// TIA Portal V17 export
// export: Created 2023-12-22T15:05:34.1188852Z, ExportSetting WithDefaults, DisplayName Totally Integrated Automation Portal, DisplayVersion V17, DisplayName TIA Portal Openness, DisplayVersion V17, DisplayName TIA Portal Version Control Interface, DisplayVersion V17, DisplayName STEP 7 Professional, DisplayVersion V17, DisplayName STEP 7 Safety, DisplayVersion V17, DisplayName WinCC Advanced, DisplayVersion V17
DATA_BLOCK "DB_OUT"   // DB102
{ S7_Optimized_Access := 'FALSE' }
VERSION : 0.1
// stored: AutoNumber false, DBAccessibleFromOPCUA true, IsOnlyStoredInLoadMemory false, IsWriteProtectedInAS false
   VAR
      AI_FT_007 { S7_SetPoint := 'True'} : "Out_AI";
      AI_FT_008 { S7_SetPoint := 'True'} : "Out_AI";
      AI_FT_009 { S7_SetPoint := 'True'} : "Out_AI";
      AI_FT_010 { S7_SetPoint := 'True'} : "Out_AI";
      AI_LT_014 { S7_SetPoint := 'True'} : "Out_AI";
      AI_LT_015 { S7_SetPoint := 'True'} : "Out_AI";
      AI_LT_016 { S7_SetPoint := 'True'} : "Out_AI";
      AI_LT_019 { S7_SetPoint := 'True'} : "Out_AI";
      AI_PT_001 { S7_SetPoint := 'True'} : "Out_AI";
      AI_PT_002 { S7_SetPoint := 'True'} : "Out_AI";
      AI_PT_003 { S7_SetPoint := 'True'} : "Out_AI";
      AI_PT_004 { S7_SetPoint := 'True'} : "Out_AI";
      AI_PT_005 { S7_SetPoint := 'True'} : "Out_AI";
      AI_PT_006 { S7_SetPoint := 'True'} : "Out_AI";
      Z_GVM_020 { S7_SetPoint := 'True'} : "Out_Z";
      Z_GVM_021 { S7_SetPoint := 'True'} : "Out_Z";
      Z_GVM_022 { S7_SetPoint := 'True'} : "Out_Z";
      Z_GCM_023 { S7_SetPoint := 'True'} : "Out_Z";
      Z_GCM_024 { S7_SetPoint := 'True'} : "Out_Z";
      Z_GCM_025 { S7_SetPoint := 'True'} : "Out_Z";
      XVS_026 { S7_SetPoint := 'True'} : "InOut_DO";
      XVS_027 { S7_SetPoint := 'True'} : "InOut_DO";
      XVS_028 { S7_SetPoint := 'True'} : "InOut_DO";
      XVS_029 { S7_SetPoint := 'True'} : "InOut_DO";
      XVS_030 { S7_SetPoint := 'True'} : "InOut_DO";
      XVS_031 { S7_SetPoint := 'True'} : "InOut_DO";
      XVS_032 { S7_SetPoint := 'True'} : "InOut_DO";
      XVS_033 { S7_SetPoint := 'True'} : "InOut_DO";
      XVS_034 { S7_SetPoint := 'True'} : "InOut_DO";
      M6_M_K_1_1 { S7_SetPoint := 'True'} : "Out_MD";
      M7_M_K_1_2 { S7_SetPoint := 'True'} : "Out_MD";
      M8_M_K_1_3 { S7_SetPoint := 'True'} : "Out_MD";
      M11_M_K_2_1 { S7_SetPoint := 'True'} : "Out_MD";
      M12_M_K_2_2 { S7_SetPoint := 'True'} : "Out_MD";
      M13_M_K_2_3 { S7_SetPoint := 'True'} : "Out_MD";
      M9_SD { S7_SetPoint := 'True'} : "Out_MDA";
      M10_Vibro { S7_SetPoint := 'True'} : "Out_MD";
      M1_BK_1 { S7_SetPoint := 'True'} : "Out_MDA";
      M2_KK_1_1 { S7_SetPoint := 'True'} : "Out_MDA";
      M3_KK_1_2 { S7_SetPoint := 'True'} : "Out_MDA";
      M4_ND_KK_1_1 { S7_SetPoint := 'True'} : "Out_MDA";
      M5_ND_KK_1_2 { S7_SetPoint := 'True'} : "Out_MDA";
      M14_ND_K_1_1 { S7_SetPoint := 'True'} : "Out_MDA";
      M15_ND_K_1_2 { S7_SetPoint := 'True'} : "Out_MDA";
      M16_ND_K_1_3 { S7_SetPoint := 'True'} : "Out_MDA";
      M17_ND_K_2_1 { S7_SetPoint := 'True'} : "Out_MDA";
      M18_ND_K_2_2 { S7_SetPoint := 'True'} : "Out_MDA";
      M19_ND_K_2_3 { S7_SetPoint := 'True'} : "Out_MDA";
      DIx : Struct
         LS_017 : Bool := FALSE;
         LS_018 : Bool := TRUE;
         FIS_011 : Bool := FALSE;
         FIS_012 : Bool := FALSE;
         FIS_013 : Bool := FALSE;
         ALS_1 : Bool := FALSE;
         ALS_2 : Bool := FALSE;
         LOCAL { S7_SetPoint := 'True'} : Bool := FALSE;
         All_Block : Bool := FALSE;
         Start_1 : Bool := FALSE;
         Start_2 : Bool := FALSE;
         Start_3 : Bool := FALSE;
         LS_019 : Bool := FALSE;
      END_STRUCT;
      PolyMix_1 : Struct
         Start : Bool := FALSE;
         SP_C : Real := 0.0;
         Messages : Struct
            Flow_Dry_Run : Bool := FALSE;
            Flow_Low : Bool := FALSE;
            LE_NoChange : Bool := FALSE;
            LE_Low : Bool := FALSE;
            LE_High : Bool := FALSE;
            LS_Low : Bool := FALSE;
            LS_NoProduct : Bool := FALSE;
            LS_Filter : Bool := FALSE;
            SD_Low : Bool := FALSE;
            Low_Weight : Bool := FALSE;
            Link_Error : Bool := FALSE;
            Alarm : Word := 16#0000;
         END_STRUCT;
      END_STRUCT;
      PolyMix_2 : Struct
         Start : Bool := FALSE;
         SP_C : Real := 0.0;
         Messages : Struct
            Flow_Dry_Run : Bool := FALSE;
            Flow_Low : Bool := FALSE;
            LE_NoChange : Bool := FALSE;
            LE_Low : Bool := FALSE;
            LE_High : Bool := FALSE;
            LS_Low : Bool := FALSE;
            LS_NoProduct : Bool := FALSE;
            LS_Filter : Bool := FALSE;
            SD_Low : Bool := FALSE;
            Low_Weight : Bool := FALSE;
            Link_Error : Bool := FALSE;
            Alarm : Word := 16#0000;
         END_STRUCT;
      END_STRUCT;
      XVS_035 { S7_SetPoint := 'True'} : "InOut_DO";
      XVS_036 { S7_SetPoint := 'True'} : "InOut_DO";
      gsm3_PolyMix_1 { S7_SetPoint := 'True'} : Real := 1.09;
      gsm3_PolyMix_2 : Real := 1.072;
      F1_Clean_Now : Bool := FALSE;
      F2_Clean_Now : Bool := FALSE;
      ALARM_NO_AIR : Bool := FALSE;
      Z_GVM_x { S7_SetPoint := 'True'} : "Out_Z";
      M_Vent : "Out_MD";
      Any_Alarms : Word := 16#0000;
      Events : Word := 16#0000;
      Lines : Array[1..7] of Struct
         Alarms : Word;
      END_STRUCT;
      res_5 : Word := 16#0000;
      res_6 : Word := 16#0000;
      res_7 : Word := 16#0000;
      res_8 : Word := 16#0000;
      res_9 : Word := 16#0000;
      res_10 : Word := 16#0000;
      Time_DTL { S7_SetPoint := 'True'} : DTL := DTL#2020-06-25-13:08:09.170187013;
   END_VAR
BEGIN
   AI_FT_007.Result := 0.04701968;
   AI_FT_007.Converter.Min_Out := 0.0;
   AI_FT_007.Converter.Max_Out := 1000.0;
   AI_FT_007.Alarms := 16#0000;
   AI_FT_007.SP.HH := 320.0;
   AI_FT_007.SP.H := 300.0;
   AI_FT_007.SP.L := 200.0;
   AI_FT_007.SP.LL := 75.0;
   AI_FT_008.Result := 0.02821181;
   AI_FT_008.Converter.Min_Out := 0.0;
   AI_FT_008.Converter.Max_Out := 100.0;
   AI_FT_008.Alarms := 16#0000;
   AI_FT_008.SP.HH := 100.0;
   AI_FT_008.SP.H := 15.0;
   AI_FT_008.SP.L := 0.5;
   AI_FT_008.SP.LL := -0.1;
   AI_FT_009.Result := 0.003616898;
   AI_FT_009.Converter.Min_Out := 0.0;
   AI_FT_009.Converter.Max_Out := 100.0;
   AI_FT_009.Alarms := 16#0000;
   AI_FT_009.SP.HH := 30.0;
   AI_FT_009.SP.H := 15.0;
   AI_FT_009.SP.L := 0.5;
   AI_FT_009.SP.LL := -0.1;
   AI_FT_010.Result := 0.01989294;
   AI_FT_010.Converter.Min_Out := 0.0;
   AI_FT_010.Converter.Max_Out := 100.0;
   AI_FT_010.Alarms := 16#0000;
   AI_FT_010.SP.HH := 50.0;
   AI_FT_010.SP.H := 40.0;
   AI_FT_010.SP.L := 0.5;
   AI_FT_010.SP.LL := -0.5;
   AI_LT_014.Result := 953.6309;
   AI_LT_014.Converter.Min_Out := 0.0;
   AI_LT_014.Converter.Max_Out := 2605.0;
   AI_LT_014.Alarms := 16#0000;
   AI_LT_014.SP.HH := 2400.0;
   AI_LT_014.SP.H := 2300.0;
   AI_LT_014.SP.L := 400.0;
   AI_LT_014.SP.LL := 220.0;
   AI_LT_015.Result := 2297.691;
   AI_LT_015.Converter.Min_Out := 0.0;
   AI_LT_015.Converter.Max_Out := 2605.0;
   AI_LT_015.Alarms := 16#0000;
   AI_LT_015.SP.HH := 2400.0;
   AI_LT_015.SP.H := 2300.0;
   AI_LT_015.SP.L := 400.0;
   AI_LT_015.SP.LL := 220.0;
   AI_LT_016.Result := 985.5756;
   AI_LT_016.Converter.Min_Out := 0.0;
   AI_LT_016.Converter.Max_Out := 1268.0;
   AI_LT_016.Alarms := 16#0004;
   AI_LT_016.SP.HH := 1060.0;
   AI_LT_016.SP.H := 950.0;
   AI_LT_016.SP.L := 250.0;
   AI_LT_016.SP.LL := 120.0;
   AI_LT_019.Result := 916.5906;
   AI_LT_019.Converter.Min_Out := 0.0;
   AI_LT_019.Converter.Max_Out := 1268.0;
   AI_LT_019.Alarms := 16#0000;
   AI_LT_019.SP.HH := 1060.0;
   AI_LT_019.SP.H := 950.0;
   AI_LT_019.SP.L := 250.0;
   AI_LT_019.SP.LL := 120.0;
   AI_PT_001.Result := 0.02823567;
   AI_PT_001.Converter.Min_Out := 0.0;
   AI_PT_001.Converter.Max_Out := 0.6;
   AI_PT_001.Alarms := 16#0000;
   AI_PT_001.SP.HH := 0.35;
   AI_PT_001.SP.H := 0.3;
   AI_PT_001.SP.L := 0.02;
   AI_PT_001.SP.LL := 0.01;
   AI_PT_002.Result := 0.02846354;
   AI_PT_002.Converter.Min_Out := 0.0;
   AI_PT_002.Converter.Max_Out := 0.6;
   AI_PT_002.Alarms := 16#0000;
   AI_PT_002.SP.HH := 0.35;
   AI_PT_002.SP.H := 0.3;
   AI_PT_002.SP.L := 0.02;
   AI_PT_002.SP.LL := 0.01;
   AI_PT_003.Result := 0.02719184;
   AI_PT_003.Converter.Min_Out := 0.0;
   AI_PT_003.Converter.Max_Out := 0.6;
   AI_PT_003.Alarms := 16#0000;
   AI_PT_003.SP.HH := 0.35;
   AI_PT_003.SP.H := 0.3;
   AI_PT_003.SP.L := 0.02;
   AI_PT_003.SP.LL := 0.01;
   AI_PT_004.Result := 0.02914063;
   AI_PT_004.Converter.Min_Out := 0.0;
   AI_PT_004.Converter.Max_Out := 0.6;
   AI_PT_004.Alarms := 16#0000;
   AI_PT_004.SP.HH := 0.35;
   AI_PT_004.SP.H := 0.3;
   AI_PT_004.SP.L := 0.02;
   AI_PT_004.SP.LL := 0.01;
   AI_PT_005.Result := 0.02641927;
   AI_PT_005.Converter.Min_Out := 0.0;
   AI_PT_005.Converter.Max_Out := 0.6;
   AI_PT_005.Alarms := 16#0000;
   AI_PT_005.SP.HH := 0.35;
   AI_PT_005.SP.H := 0.3;
   AI_PT_005.SP.L := 0.02;
   AI_PT_005.SP.LL := 0.01;
   AI_PT_006.Result := 0.02695746;
   AI_PT_006.Converter.Min_Out := 0.0;
   AI_PT_006.Converter.Max_Out := 0.6;
   AI_PT_006.Alarms := 16#0000;
   AI_PT_006.SP.HH := 0.35;
   AI_PT_006.SP.H := 0.3;
   AI_PT_006.SP.L := 0.02;
   AI_PT_006.SP.LL := 0.01;
   Z_GVM_020.CMD.Hand := FALSE;
   Z_GVM_020.CMD.Start_A := FALSE;
   Z_GVM_020.CMD.Start_M := FALSE;
   Z_GVM_020.CMD.Force := FALSE;
   Z_GVM_020.CMD.Lock := FALSE;
   Z_GVM_020.CMD.Local := FALSE;
   Z_GVM_020.CMD.Service := FALSE;
   Z_GVM_020.CMD.Safety := FALSE;
   Z_GVM_020.CMD.Alarm := FALSE;
   Z_GVM_020.CMD.Reset := FALSE;
   Z_GVM_020.CMD.Sim := FALSE;
   Z_GVM_020.CMD.Vector := FALSE;
   Z_GVM_020.CMD.Ready := FALSE;
   Z_GVM_020.CMD.Resourse := FALSE;
   Z_GVM_020.Status := 0;
   Z_GVM_020.T_ON := 12;
   Z_GVM_020.T_OFF := 12;
   Z_GVM_020.Alarms := 16#0000;
   Z_GVM_021.CMD.Hand := FALSE;
   Z_GVM_021.CMD.Start_A := FALSE;
   Z_GVM_021.CMD.Start_M := FALSE;
   Z_GVM_021.CMD.Force := FALSE;
   Z_GVM_021.CMD.Lock := FALSE;
   Z_GVM_021.CMD.Local := FALSE;
   Z_GVM_021.CMD.Service := FALSE;
   Z_GVM_021.CMD.Safety := FALSE;
   Z_GVM_021.CMD.Alarm := FALSE;
   Z_GVM_021.CMD.Reset := FALSE;
   Z_GVM_021.CMD.Sim := FALSE;
   Z_GVM_021.CMD.Vector := FALSE;
   Z_GVM_021.CMD.Ready := FALSE;
   Z_GVM_021.CMD.Resourse := FALSE;
   Z_GVM_021.Status := 0;
   Z_GVM_021.T_ON := 12;
   Z_GVM_021.T_OFF := 12;
   Z_GVM_021.Alarms := 16#0000;
   Z_GVM_022.CMD.Hand := FALSE;
   Z_GVM_022.CMD.Start_A := FALSE;
   Z_GVM_022.CMD.Start_M := FALSE;
   Z_GVM_022.CMD.Force := FALSE;
   Z_GVM_022.CMD.Lock := FALSE;
   Z_GVM_022.CMD.Local := FALSE;
   Z_GVM_022.CMD.Service := FALSE;
   Z_GVM_022.CMD.Safety := FALSE;
   Z_GVM_022.CMD.Alarm := FALSE;
   Z_GVM_022.CMD.Reset := FALSE;
   Z_GVM_022.CMD.Sim := FALSE;
   Z_GVM_022.CMD.Vector := FALSE;
   Z_GVM_022.CMD.Ready := FALSE;
   Z_GVM_022.CMD.Resourse := FALSE;
   Z_GVM_022.Status := 0;
   Z_GVM_022.T_ON := 12;
   Z_GVM_022.T_OFF := 12;
   Z_GVM_022.Alarms := 16#0000;
   Z_GCM_023.CMD.Hand := FALSE;
   Z_GCM_023.CMD.Start_A := FALSE;
   Z_GCM_023.CMD.Start_M := FALSE;
   Z_GCM_023.CMD.Force := FALSE;
   Z_GCM_023.CMD.Lock := FALSE;
   Z_GCM_023.CMD.Local := FALSE;
   Z_GCM_023.CMD.Service := FALSE;
   Z_GCM_023.CMD.Safety := FALSE;
   Z_GCM_023.CMD.Alarm := FALSE;
   Z_GCM_023.CMD.Reset := FALSE;
   Z_GCM_023.CMD.Sim := FALSE;
   Z_GCM_023.CMD.Vector := FALSE;
   Z_GCM_023.CMD.Ready := FALSE;
   Z_GCM_023.CMD.Resourse := FALSE;
   Z_GCM_023.Status := 0;
   Z_GCM_023.T_ON := 12;
   Z_GCM_023.T_OFF := 12;
   Z_GCM_023.Alarms := 16#0000;
   Z_GCM_024.CMD.Hand := FALSE;
   Z_GCM_024.CMD.Start_A := FALSE;
   Z_GCM_024.CMD.Start_M := FALSE;
   Z_GCM_024.CMD.Force := FALSE;
   Z_GCM_024.CMD.Lock := FALSE;
   Z_GCM_024.CMD.Local := FALSE;
   Z_GCM_024.CMD.Service := FALSE;
   Z_GCM_024.CMD.Safety := FALSE;
   Z_GCM_024.CMD.Alarm := FALSE;
   Z_GCM_024.CMD.Reset := FALSE;
   Z_GCM_024.CMD.Sim := FALSE;
   Z_GCM_024.CMD.Vector := FALSE;
   Z_GCM_024.CMD.Ready := FALSE;
   Z_GCM_024.CMD.Resourse := FALSE;
   Z_GCM_024.Status := 0;
   Z_GCM_024.T_ON := 12;
   Z_GCM_024.T_OFF := 12;
   Z_GCM_024.Alarms := 16#0000;
   Z_GCM_025.CMD.Hand := FALSE;
   Z_GCM_025.CMD.Start_A := FALSE;
   Z_GCM_025.CMD.Start_M := FALSE;
   Z_GCM_025.CMD.Force := FALSE;
   Z_GCM_025.CMD.Lock := FALSE;
   Z_GCM_025.CMD.Local := FALSE;
   Z_GCM_025.CMD.Service := FALSE;
   Z_GCM_025.CMD.Safety := FALSE;
   Z_GCM_025.CMD.Alarm := FALSE;
   Z_GCM_025.CMD.Reset := FALSE;
   Z_GCM_025.CMD.Sim := FALSE;
   Z_GCM_025.CMD.Vector := FALSE;
   Z_GCM_025.CMD.Ready := FALSE;
   Z_GCM_025.CMD.Resourse := FALSE;
   Z_GCM_025.Status := 0;
   Z_GCM_025.T_ON := 12;
   Z_GCM_025.T_OFF := 12;
   Z_GCM_025.Alarms := 16#0000;
   XVS_026.CMD.Hand := FALSE;
   XVS_026.CMD.Start_A := FALSE;
   XVS_026.CMD.Start_M := FALSE;
   XVS_026.CMD.Force := FALSE;
   XVS_026.CMD.Lock := FALSE;
   XVS_026.CMD.Local := FALSE;
   XVS_026.CMD.Service := FALSE;
   XVS_026.CMD.Safety := FALSE;
   XVS_026.CMD.Alarm := FALSE;
   XVS_026.CMD.Reset := FALSE;
   XVS_026.CMD.Sim := FALSE;
   XVS_026.CMD.Vector := FALSE;
   XVS_026.CMD.Ready := FALSE;
   XVS_026.CMD.Resourse := FALSE;
   XVS_027.CMD.Hand := FALSE;
   XVS_027.CMD.Start_A := FALSE;
   XVS_027.CMD.Start_M := FALSE;
   XVS_027.CMD.Force := FALSE;
   XVS_027.CMD.Lock := FALSE;
   XVS_027.CMD.Local := FALSE;
   XVS_027.CMD.Service := FALSE;
   XVS_027.CMD.Safety := FALSE;
   XVS_027.CMD.Alarm := FALSE;
   XVS_027.CMD.Reset := FALSE;
   XVS_027.CMD.Sim := FALSE;
   XVS_027.CMD.Vector := FALSE;
   XVS_027.CMD.Ready := FALSE;
   XVS_027.CMD.Resourse := FALSE;
   XVS_028.CMD.Hand := FALSE;
   XVS_028.CMD.Start_A := FALSE;
   XVS_028.CMD.Start_M := FALSE;
   XVS_028.CMD.Force := FALSE;
   XVS_028.CMD.Lock := FALSE;
   XVS_028.CMD.Local := FALSE;
   XVS_028.CMD.Service := FALSE;
   XVS_028.CMD.Safety := FALSE;
   XVS_028.CMD.Alarm := FALSE;
   XVS_028.CMD.Reset := FALSE;
   XVS_028.CMD.Sim := FALSE;
   XVS_028.CMD.Vector := FALSE;
   XVS_028.CMD.Ready := FALSE;
   XVS_028.CMD.Resourse := FALSE;
   XVS_029.CMD.Hand := FALSE;
   XVS_029.CMD.Start_A := FALSE;
   XVS_029.CMD.Start_M := FALSE;
   XVS_029.CMD.Force := FALSE;
   XVS_029.CMD.Lock := FALSE;
   XVS_029.CMD.Local := FALSE;
   XVS_029.CMD.Service := FALSE;
   XVS_029.CMD.Safety := FALSE;
   XVS_029.CMD.Alarm := FALSE;
   XVS_029.CMD.Reset := FALSE;
   XVS_029.CMD.Sim := FALSE;
   XVS_029.CMD.Vector := FALSE;
   XVS_029.CMD.Ready := FALSE;
   XVS_029.CMD.Resourse := FALSE;
   XVS_030.CMD.Hand := FALSE;
   XVS_030.CMD.Start_A := FALSE;
   XVS_030.CMD.Start_M := FALSE;
   XVS_030.CMD.Force := FALSE;
   XVS_030.CMD.Lock := FALSE;
   XVS_030.CMD.Local := FALSE;
   XVS_030.CMD.Service := FALSE;
   XVS_030.CMD.Safety := FALSE;
   XVS_030.CMD.Alarm := FALSE;
   XVS_030.CMD.Reset := FALSE;
   XVS_030.CMD.Sim := FALSE;
   XVS_030.CMD.Vector := FALSE;
   XVS_030.CMD.Ready := FALSE;
   XVS_030.CMD.Resourse := FALSE;
   XVS_031.CMD.Hand := FALSE;
   XVS_031.CMD.Start_A := FALSE;
   XVS_031.CMD.Start_M := FALSE;
   XVS_031.CMD.Force := FALSE;
   XVS_031.CMD.Lock := FALSE;
   XVS_031.CMD.Local := FALSE;
   XVS_031.CMD.Service := FALSE;
   XVS_031.CMD.Safety := FALSE;
   XVS_031.CMD.Alarm := FALSE;
   XVS_031.CMD.Reset := FALSE;
   XVS_031.CMD.Sim := FALSE;
   XVS_031.CMD.Vector := FALSE;
   XVS_031.CMD.Ready := FALSE;
   XVS_031.CMD.Resourse := FALSE;
   XVS_032.CMD.Hand := FALSE;
   XVS_032.CMD.Start_A := FALSE;
   XVS_032.CMD.Start_M := FALSE;
   XVS_032.CMD.Force := FALSE;
   XVS_032.CMD.Lock := FALSE;
   XVS_032.CMD.Local := FALSE;
   XVS_032.CMD.Service := FALSE;
   XVS_032.CMD.Safety := FALSE;
   XVS_032.CMD.Alarm := FALSE;
   XVS_032.CMD.Reset := FALSE;
   XVS_032.CMD.Sim := FALSE;
   XVS_032.CMD.Vector := FALSE;
   XVS_032.CMD.Ready := FALSE;
   XVS_032.CMD.Resourse := FALSE;
   XVS_033.CMD.Hand := FALSE;
   XVS_033.CMD.Start_A := FALSE;
   XVS_033.CMD.Start_M := FALSE;
   XVS_033.CMD.Force := FALSE;
   XVS_033.CMD.Lock := FALSE;
   XVS_033.CMD.Local := FALSE;
   XVS_033.CMD.Service := FALSE;
   XVS_033.CMD.Safety := FALSE;
   XVS_033.CMD.Alarm := FALSE;
   XVS_033.CMD.Reset := FALSE;
   XVS_033.CMD.Sim := FALSE;
   XVS_033.CMD.Vector := FALSE;
   XVS_033.CMD.Ready := FALSE;
   XVS_033.CMD.Resourse := FALSE;
   XVS_034.CMD.Hand := FALSE;
   XVS_034.CMD.Start_A := FALSE;
   XVS_034.CMD.Start_M := FALSE;
   XVS_034.CMD.Force := FALSE;
   XVS_034.CMD.Lock := FALSE;
   XVS_034.CMD.Local := FALSE;
   XVS_034.CMD.Service := FALSE;
   XVS_034.CMD.Safety := FALSE;
   XVS_034.CMD.Alarm := FALSE;
   XVS_034.CMD.Reset := FALSE;
   XVS_034.CMD.Sim := FALSE;
   XVS_034.CMD.Vector := FALSE;
   XVS_034.CMD.Ready := FALSE;
   XVS_034.CMD.Resourse := FALSE;
   M6_M_K_1_1.CMD.Hand := FALSE;
   M6_M_K_1_1.CMD.Start_A := TRUE;
   M6_M_K_1_1.CMD.Start_M := TRUE;
   M6_M_K_1_1.CMD.Force := FALSE;
   M6_M_K_1_1.CMD.Lock := FALSE;
   M6_M_K_1_1.CMD.Local := FALSE;
   M6_M_K_1_1.CMD.Service := FALSE;
   M6_M_K_1_1.CMD.Safety := FALSE;
   M6_M_K_1_1.CMD.Alarm := FALSE;
   M6_M_K_1_1.CMD.Reset := FALSE;
   M6_M_K_1_1.CMD.Sim := FALSE;
   M6_M_K_1_1.CMD.Vector := FALSE;
   M6_M_K_1_1.CMD.Ready := FALSE;
   M6_M_K_1_1.CMD.Resourse := FALSE;
   M6_M_K_1_1.Status := 1;
   M6_M_K_1_1.T_ON := 2;
   M6_M_K_1_1.T_OFF := 2;
   M6_M_K_1_1.Alarms := 16#0000;
   M6_M_K_1_1.Res_h := 271;
   M7_M_K_1_2.CMD.Hand := FALSE;
   M7_M_K_1_2.CMD.Start_A := TRUE;
   M7_M_K_1_2.CMD.Start_M := TRUE;
   M7_M_K_1_2.CMD.Force := FALSE;
   M7_M_K_1_2.CMD.Lock := FALSE;
   M7_M_K_1_2.CMD.Local := FALSE;
   M7_M_K_1_2.CMD.Service := FALSE;
   M7_M_K_1_2.CMD.Safety := FALSE;
   M7_M_K_1_2.CMD.Alarm := FALSE;
   M7_M_K_1_2.CMD.Reset := FALSE;
   M7_M_K_1_2.CMD.Sim := FALSE;
   M7_M_K_1_2.CMD.Vector := FALSE;
   M7_M_K_1_2.CMD.Ready := FALSE;
   M7_M_K_1_2.CMD.Resourse := FALSE;
   M7_M_K_1_2.Status := 1;
   M7_M_K_1_2.T_ON := 2;
   M7_M_K_1_2.T_OFF := 2;
   M7_M_K_1_2.Alarms := 16#0000;
   M7_M_K_1_2.Res_h := 133;
   M8_M_K_1_3.CMD.Hand := FALSE;
   M8_M_K_1_3.CMD.Start_A := TRUE;
   M8_M_K_1_3.CMD.Start_M := TRUE;
   M8_M_K_1_3.CMD.Force := FALSE;
   M8_M_K_1_3.CMD.Lock := FALSE;
   M8_M_K_1_3.CMD.Local := FALSE;
   M8_M_K_1_3.CMD.Service := FALSE;
   M8_M_K_1_3.CMD.Safety := FALSE;
   M8_M_K_1_3.CMD.Alarm := FALSE;
   M8_M_K_1_3.CMD.Reset := FALSE;
   M8_M_K_1_3.CMD.Sim := FALSE;
   M8_M_K_1_3.CMD.Vector := FALSE;
   M8_M_K_1_3.CMD.Ready := FALSE;
   M8_M_K_1_3.CMD.Resourse := FALSE;
   M8_M_K_1_3.Status := 1;
   M8_M_K_1_3.T_ON := 2;
   M8_M_K_1_3.T_OFF := 2;
   M8_M_K_1_3.Alarms := 16#0000;
   M8_M_K_1_3.Res_h := 269;
   M11_M_K_2_1.CMD.Hand := FALSE;
   M11_M_K_2_1.CMD.Start_A := FALSE;
   M11_M_K_2_1.CMD.Start_M := FALSE;
   M11_M_K_2_1.CMD.Force := FALSE;
   M11_M_K_2_1.CMD.Lock := FALSE;
   M11_M_K_2_1.CMD.Local := FALSE;
   M11_M_K_2_1.CMD.Service := FALSE;
   M11_M_K_2_1.CMD.Safety := FALSE;
   M11_M_K_2_1.CMD.Alarm := FALSE;
   M11_M_K_2_1.CMD.Reset := FALSE;
   M11_M_K_2_1.CMD.Sim := FALSE;
   M11_M_K_2_1.CMD.Vector := FALSE;
   M11_M_K_2_1.CMD.Ready := FALSE;
   M11_M_K_2_1.CMD.Resourse := FALSE;
   M11_M_K_2_1.Status := 0;
   M11_M_K_2_1.T_ON := 2;
   M11_M_K_2_1.T_OFF := 2;
   M11_M_K_2_1.Alarms := 16#0000;
   M11_M_K_2_1.Res_h := 227;
   M12_M_K_2_2.CMD.Hand := FALSE;
   M12_M_K_2_2.CMD.Start_A := FALSE;
   M12_M_K_2_2.CMD.Start_M := FALSE;
   M12_M_K_2_2.CMD.Force := FALSE;
   M12_M_K_2_2.CMD.Lock := FALSE;
   M12_M_K_2_2.CMD.Local := FALSE;
   M12_M_K_2_2.CMD.Service := FALSE;
   M12_M_K_2_2.CMD.Safety := FALSE;
   M12_M_K_2_2.CMD.Alarm := FALSE;
   M12_M_K_2_2.CMD.Reset := FALSE;
   M12_M_K_2_2.CMD.Sim := FALSE;
   M12_M_K_2_2.CMD.Vector := FALSE;
   M12_M_K_2_2.CMD.Ready := FALSE;
   M12_M_K_2_2.CMD.Resourse := FALSE;
   M12_M_K_2_2.Status := 0;
   M12_M_K_2_2.T_ON := 2;
   M12_M_K_2_2.T_OFF := 2;
   M12_M_K_2_2.Alarms := 16#0000;
   M12_M_K_2_2.Res_h := 182;
   M13_M_K_2_3.CMD.Hand := FALSE;
   M13_M_K_2_3.CMD.Start_A := FALSE;
   M13_M_K_2_3.CMD.Start_M := FALSE;
   M13_M_K_2_3.CMD.Force := FALSE;
   M13_M_K_2_3.CMD.Lock := FALSE;
   M13_M_K_2_3.CMD.Local := FALSE;
   M13_M_K_2_3.CMD.Service := FALSE;
   M13_M_K_2_3.CMD.Safety := FALSE;
   M13_M_K_2_3.CMD.Alarm := FALSE;
   M13_M_K_2_3.CMD.Reset := FALSE;
   M13_M_K_2_3.CMD.Sim := FALSE;
   M13_M_K_2_3.CMD.Vector := FALSE;
   M13_M_K_2_3.CMD.Ready := FALSE;
   M13_M_K_2_3.CMD.Resourse := FALSE;
   M13_M_K_2_3.Status := 0;
   M13_M_K_2_3.T_ON := 2;
   M13_M_K_2_3.T_OFF := 2;
   M13_M_K_2_3.Alarms := 16#0000;
   M13_M_K_2_3.Res_h := 163;
   M9_SD.CMD.Hand := FALSE;
   M9_SD.CMD.Start_A := FALSE;
   M9_SD.CMD.Start_M := FALSE;
   M9_SD.CMD.Force := FALSE;
   M9_SD.CMD.Lock := FALSE;
   M9_SD.CMD.Local := FALSE;
   M9_SD.CMD.Service := FALSE;
   M9_SD.CMD.Safety := FALSE;
   M9_SD.CMD.Alarm := FALSE;
   M9_SD.CMD.Reset := FALSE;
   M9_SD.CMD.Sim := FALSE;
   M9_SD.CMD.Vector := FALSE;
   M9_SD.CMD.Ready := FALSE;
   M9_SD.CMD.Resourse := FALSE;
   M9_SD.Status := 0;
   M9_SD.T_ON := 2;
   M9_SD.T_OFF := 2;
   M9_SD.Alarms := 16#0000;
   M9_SD.Res_h := 26;
   M9_SD.SP_M := 0.0;
   M9_SD.Converter.Min_Out := 0.0;
   M9_SD.Converter.Max_Out := 100.0;
   M10_Vibro.CMD.Hand := FALSE;
   M10_Vibro.CMD.Start_A := FALSE;
   M10_Vibro.CMD.Start_M := FALSE;
   M10_Vibro.CMD.Force := FALSE;
   M10_Vibro.CMD.Lock := FALSE;
   M10_Vibro.CMD.Local := FALSE;
   M10_Vibro.CMD.Service := FALSE;
   M10_Vibro.CMD.Safety := FALSE;
   M10_Vibro.CMD.Alarm := FALSE;
   M10_Vibro.CMD.Reset := FALSE;
   M10_Vibro.CMD.Sim := FALSE;
   M10_Vibro.CMD.Vector := FALSE;
   M10_Vibro.CMD.Ready := FALSE;
   M10_Vibro.CMD.Resourse := FALSE;
   M10_Vibro.Status := 0;
   M10_Vibro.T_ON := 2;
   M10_Vibro.T_OFF := 2;
   M10_Vibro.Alarms := 16#0000;
   M10_Vibro.Res_h := 0;
   M1_BK_1.CMD.Hand := FALSE;
   M1_BK_1.CMD.Start_A := FALSE;
   M1_BK_1.CMD.Start_M := FALSE;
   M1_BK_1.CMD.Force := FALSE;
   M1_BK_1.CMD.Lock := TRUE;
   M1_BK_1.CMD.Local := FALSE;
   M1_BK_1.CMD.Service := FALSE;
   M1_BK_1.CMD.Safety := FALSE;
   M1_BK_1.CMD.Alarm := FALSE;
   M1_BK_1.CMD.Reset := FALSE;
   M1_BK_1.CMD.Sim := FALSE;
   M1_BK_1.CMD.Vector := FALSE;
   M1_BK_1.CMD.Ready := FALSE;
   M1_BK_1.CMD.Resourse := FALSE;
   M1_BK_1.Status := 0;
   M1_BK_1.T_ON := 2;
   M1_BK_1.T_OFF := 2;
   M1_BK_1.Alarms := 16#0000;
   M1_BK_1.Res_h := 2;
   M1_BK_1.SP_M := 100.0;
   M1_BK_1.Converter.Min_Out := 0.0;
   M1_BK_1.Converter.Max_Out := 0.0;
   M2_KK_1_1.CMD.Hand := FALSE;
   M2_KK_1_1.CMD.Start_A := FALSE;
   M2_KK_1_1.CMD.Start_M := FALSE;
   M2_KK_1_1.CMD.Force := FALSE;
   M2_KK_1_1.CMD.Lock := TRUE;
   M2_KK_1_1.CMD.Local := FALSE;
   M2_KK_1_1.CMD.Service := FALSE;
   M2_KK_1_1.CMD.Safety := FALSE;
   M2_KK_1_1.CMD.Alarm := FALSE;
   M2_KK_1_1.CMD.Reset := FALSE;
   M2_KK_1_1.CMD.Sim := FALSE;
   M2_KK_1_1.CMD.Vector := FALSE;
   M2_KK_1_1.CMD.Ready := FALSE;
   M2_KK_1_1.CMD.Resourse := FALSE;
   M2_KK_1_1.Status := 0;
   M2_KK_1_1.T_ON := 2;
   M2_KK_1_1.T_OFF := 2;
   M2_KK_1_1.Alarms := 16#0000;
   M2_KK_1_1.Res_h := 2;
   M2_KK_1_1.SP_M := 0.0;
   M2_KK_1_1.Converter.Min_Out := 0.0;
   M2_KK_1_1.Converter.Max_Out := 0.0;
   M3_KK_1_2.CMD.Hand := FALSE;
   M3_KK_1_2.CMD.Start_A := FALSE;
   M3_KK_1_2.CMD.Start_M := FALSE;
   M3_KK_1_2.CMD.Force := FALSE;
   M3_KK_1_2.CMD.Lock := TRUE;
   M3_KK_1_2.CMD.Local := FALSE;
   M3_KK_1_2.CMD.Service := FALSE;
   M3_KK_1_2.CMD.Safety := FALSE;
   M3_KK_1_2.CMD.Alarm := FALSE;
   M3_KK_1_2.CMD.Reset := FALSE;
   M3_KK_1_2.CMD.Sim := FALSE;
   M3_KK_1_2.CMD.Vector := FALSE;
   M3_KK_1_2.CMD.Ready := FALSE;
   M3_KK_1_2.CMD.Resourse := FALSE;
   M3_KK_1_2.Status := 0;
   M3_KK_1_2.T_ON := 2;
   M3_KK_1_2.T_OFF := 2;
   M3_KK_1_2.Alarms := 16#0000;
   M3_KK_1_2.Res_h := 0;
   M3_KK_1_2.SP_M := 0.0;
   M3_KK_1_2.Converter.Min_Out := 0.0;
   M3_KK_1_2.Converter.Max_Out := 0.0;
   M4_ND_KK_1_1.CMD.Hand := FALSE;
   M4_ND_KK_1_1.CMD.Start_A := FALSE;
   M4_ND_KK_1_1.CMD.Start_M := FALSE;
   M4_ND_KK_1_1.CMD.Force := FALSE;
   M4_ND_KK_1_1.CMD.Lock := TRUE;
   M4_ND_KK_1_1.CMD.Local := FALSE;
   M4_ND_KK_1_1.CMD.Service := FALSE;
   M4_ND_KK_1_1.CMD.Safety := FALSE;
   M4_ND_KK_1_1.CMD.Alarm := FALSE;
   M4_ND_KK_1_1.CMD.Reset := FALSE;
   M4_ND_KK_1_1.CMD.Sim := FALSE;
   M4_ND_KK_1_1.CMD.Vector := FALSE;
   M4_ND_KK_1_1.CMD.Ready := FALSE;
   M4_ND_KK_1_1.CMD.Resourse := FALSE;
   M4_ND_KK_1_1.Status := 0;
   M4_ND_KK_1_1.T_ON := 0;
   M4_ND_KK_1_1.T_OFF := 0;
   M4_ND_KK_1_1.Alarms := 16#0000;
   M4_ND_KK_1_1.Res_h := 1;
   M4_ND_KK_1_1.SP_M := 0.0;
   M4_ND_KK_1_1.Converter.Min_Out := 0.0;
   M4_ND_KK_1_1.Converter.Max_Out := 15.6;
   M5_ND_KK_1_2.CMD.Hand := FALSE;
   M5_ND_KK_1_2.CMD.Start_A := FALSE;
   M5_ND_KK_1_2.CMD.Start_M := FALSE;
   M5_ND_KK_1_2.CMD.Force := FALSE;
   M5_ND_KK_1_2.CMD.Lock := TRUE;
   M5_ND_KK_1_2.CMD.Local := FALSE;
   M5_ND_KK_1_2.CMD.Service := FALSE;
   M5_ND_KK_1_2.CMD.Safety := FALSE;
   M5_ND_KK_1_2.CMD.Alarm := FALSE;
   M5_ND_KK_1_2.CMD.Reset := FALSE;
   M5_ND_KK_1_2.CMD.Sim := FALSE;
   M5_ND_KK_1_2.CMD.Vector := FALSE;
   M5_ND_KK_1_2.CMD.Ready := FALSE;
   M5_ND_KK_1_2.CMD.Resourse := FALSE;
   M5_ND_KK_1_2.Status := 0;
   M5_ND_KK_1_2.T_ON := 0;
   M5_ND_KK_1_2.T_OFF := 0;
   M5_ND_KK_1_2.Alarms := 16#0000;
   M5_ND_KK_1_2.Res_h := 5;
   M5_ND_KK_1_2.SP_M := 0.0;
   M5_ND_KK_1_2.Converter.Min_Out := 0.0;
   M5_ND_KK_1_2.Converter.Max_Out := 15.6;
   M14_ND_K_1_1.CMD.Hand := FALSE;
   M14_ND_K_1_1.CMD.Start_A := FALSE;
   M14_ND_K_1_1.CMD.Start_M := FALSE;
   M14_ND_K_1_1.CMD.Force := FALSE;
   M14_ND_K_1_1.CMD.Lock := FALSE;
   M14_ND_K_1_1.CMD.Local := FALSE;
   M14_ND_K_1_1.CMD.Service := FALSE;
   M14_ND_K_1_1.CMD.Safety := FALSE;
   M14_ND_K_1_1.CMD.Alarm := FALSE;
   M14_ND_K_1_1.CMD.Reset := FALSE;
   M14_ND_K_1_1.CMD.Sim := FALSE;
   M14_ND_K_1_1.CMD.Vector := FALSE;
   M14_ND_K_1_1.CMD.Ready := FALSE;
   M14_ND_K_1_1.CMD.Resourse := FALSE;
   M14_ND_K_1_1.Status := 0;
   M14_ND_K_1_1.T_ON := 0;
   M14_ND_K_1_1.T_OFF := 0;
   M14_ND_K_1_1.Alarms := 16#0000;
   M14_ND_K_1_1.Res_h := 42;
   M14_ND_K_1_1.SP_M := 0.0;
   M14_ND_K_1_1.Converter.Min_Out := 0.0;
   M14_ND_K_1_1.Converter.Max_Out := 15.6;
   M15_ND_K_1_2.CMD.Hand := FALSE;
   M15_ND_K_1_2.CMD.Start_A := FALSE;
   M15_ND_K_1_2.CMD.Start_M := FALSE;
   M15_ND_K_1_2.CMD.Force := FALSE;
   M15_ND_K_1_2.CMD.Lock := FALSE;
   M15_ND_K_1_2.CMD.Local := FALSE;
   M15_ND_K_1_2.CMD.Service := FALSE;
   M15_ND_K_1_2.CMD.Safety := FALSE;
   M15_ND_K_1_2.CMD.Alarm := FALSE;
   M15_ND_K_1_2.CMD.Reset := FALSE;
   M15_ND_K_1_2.CMD.Sim := FALSE;
   M15_ND_K_1_2.CMD.Vector := FALSE;
   M15_ND_K_1_2.CMD.Ready := FALSE;
   M15_ND_K_1_2.CMD.Resourse := FALSE;
   M15_ND_K_1_2.Status := 0;
   M15_ND_K_1_2.T_ON := 0;
   M15_ND_K_1_2.T_OFF := 0;
   M15_ND_K_1_2.Alarms := 16#0000;
   M15_ND_K_1_2.Res_h := 72;
   M15_ND_K_1_2.SP_M := 0.0;
   M15_ND_K_1_2.Converter.Min_Out := 0.0;
   M15_ND_K_1_2.Converter.Max_Out := 15.6;
   M16_ND_K_1_3.CMD.Hand := FALSE;
   M16_ND_K_1_3.CMD.Start_A := FALSE;
   M16_ND_K_1_3.CMD.Start_M := FALSE;
   M16_ND_K_1_3.CMD.Force := FALSE;
   M16_ND_K_1_3.CMD.Lock := FALSE;
   M16_ND_K_1_3.CMD.Local := FALSE;
   M16_ND_K_1_3.CMD.Service := FALSE;
   M16_ND_K_1_3.CMD.Safety := FALSE;
   M16_ND_K_1_3.CMD.Alarm := FALSE;
   M16_ND_K_1_3.CMD.Reset := FALSE;
   M16_ND_K_1_3.CMD.Sim := FALSE;
   M16_ND_K_1_3.CMD.Vector := FALSE;
   M16_ND_K_1_3.CMD.Ready := FALSE;
   M16_ND_K_1_3.CMD.Resourse := FALSE;
   M16_ND_K_1_3.Status := 0;
   M16_ND_K_1_3.T_ON := 0;
   M16_ND_K_1_3.T_OFF := 0;
   M16_ND_K_1_3.Alarms := 16#0000;
   M16_ND_K_1_3.Res_h := 11;
   M16_ND_K_1_3.SP_M := 0.0;
   M16_ND_K_1_3.Converter.Min_Out := 0.0;
   M16_ND_K_1_3.Converter.Max_Out := 15.6;
   M17_ND_K_2_1.CMD.Hand := FALSE;
   M17_ND_K_2_1.CMD.Start_A := FALSE;
   M17_ND_K_2_1.CMD.Start_M := FALSE;
   M17_ND_K_2_1.CMD.Force := FALSE;
   M17_ND_K_2_1.CMD.Lock := FALSE;
   M17_ND_K_2_1.CMD.Local := FALSE;
   M17_ND_K_2_1.CMD.Service := FALSE;
   M17_ND_K_2_1.CMD.Safety := FALSE;
   M17_ND_K_2_1.CMD.Alarm := FALSE;
   M17_ND_K_2_1.CMD.Reset := FALSE;
   M17_ND_K_2_1.CMD.Sim := FALSE;
   M17_ND_K_2_1.CMD.Vector := FALSE;
   M17_ND_K_2_1.CMD.Ready := FALSE;
   M17_ND_K_2_1.CMD.Resourse := FALSE;
   M17_ND_K_2_1.Status := 0;
   M17_ND_K_2_1.T_ON := 0;
   M17_ND_K_2_1.T_OFF := 0;
   M17_ND_K_2_1.Alarms := 16#0000;
   M17_ND_K_2_1.Res_h := 160;
   M17_ND_K_2_1.SP_M := 0.0;
   M17_ND_K_2_1.Converter.Min_Out := 0.0;
   M17_ND_K_2_1.Converter.Max_Out := 15.6;
   M18_ND_K_2_2.CMD.Hand := FALSE;
   M18_ND_K_2_2.CMD.Start_A := FALSE;
   M18_ND_K_2_2.CMD.Start_M := FALSE;
   M18_ND_K_2_2.CMD.Force := FALSE;
   M18_ND_K_2_2.CMD.Lock := FALSE;
   M18_ND_K_2_2.CMD.Local := FALSE;
   M18_ND_K_2_2.CMD.Service := FALSE;
   M18_ND_K_2_2.CMD.Safety := FALSE;
   M18_ND_K_2_2.CMD.Alarm := FALSE;
   M18_ND_K_2_2.CMD.Reset := FALSE;
   M18_ND_K_2_2.CMD.Sim := FALSE;
   M18_ND_K_2_2.CMD.Vector := FALSE;
   M18_ND_K_2_2.CMD.Ready := FALSE;
   M18_ND_K_2_2.CMD.Resourse := FALSE;
   M18_ND_K_2_2.Status := 0;
   M18_ND_K_2_2.T_ON := 0;
   M18_ND_K_2_2.T_OFF := 0;
   M18_ND_K_2_2.Alarms := 16#0000;
   M18_ND_K_2_2.Res_h := 1;
   M18_ND_K_2_2.SP_M := 0.0;
   M18_ND_K_2_2.Converter.Min_Out := 0.0;
   M18_ND_K_2_2.Converter.Max_Out := 15.6;
   M19_ND_K_2_3.CMD.Hand := FALSE;
   M19_ND_K_2_3.CMD.Start_A := FALSE;
   M19_ND_K_2_3.CMD.Start_M := FALSE;
   M19_ND_K_2_3.CMD.Force := FALSE;
   M19_ND_K_2_3.CMD.Lock := FALSE;
   M19_ND_K_2_3.CMD.Local := FALSE;
   M19_ND_K_2_3.CMD.Service := FALSE;
   M19_ND_K_2_3.CMD.Safety := FALSE;
   M19_ND_K_2_3.CMD.Alarm := FALSE;
   M19_ND_K_2_3.CMD.Reset := FALSE;
   M19_ND_K_2_3.CMD.Sim := FALSE;
   M19_ND_K_2_3.CMD.Vector := FALSE;
   M19_ND_K_2_3.CMD.Ready := FALSE;
   M19_ND_K_2_3.CMD.Resourse := FALSE;
   M19_ND_K_2_3.Status := 0;
   M19_ND_K_2_3.T_ON := 0;
   M19_ND_K_2_3.T_OFF := 0;
   M19_ND_K_2_3.Alarms := 16#0000;
   M19_ND_K_2_3.Res_h := 0;
   M19_ND_K_2_3.SP_M := 0.0;
   M19_ND_K_2_3.Converter.Min_Out := 0.0;
   M19_ND_K_2_3.Converter.Max_Out := 15.6;
   XVS_035.CMD.Hand := FALSE;
   XVS_035.CMD.Start_A := TRUE;
   XVS_035.CMD.Start_M := TRUE;
   XVS_035.CMD.Force := FALSE;
   XVS_035.CMD.Lock := FALSE;
   XVS_035.CMD.Local := FALSE;
   XVS_035.CMD.Service := FALSE;
   XVS_035.CMD.Safety := FALSE;
   XVS_035.CMD.Alarm := FALSE;
   XVS_035.CMD.Reset := FALSE;
   XVS_035.CMD.Sim := FALSE;
   XVS_035.CMD.Vector := FALSE;
   XVS_035.CMD.Ready := FALSE;
   XVS_035.CMD.Resourse := FALSE;
   XVS_036.CMD.Hand := FALSE;
   XVS_036.CMD.Start_A := TRUE;
   XVS_036.CMD.Start_M := TRUE;
   XVS_036.CMD.Force := FALSE;
   XVS_036.CMD.Lock := FALSE;
   XVS_036.CMD.Local := FALSE;
   XVS_036.CMD.Service := FALSE;
   XVS_036.CMD.Safety := FALSE;
   XVS_036.CMD.Alarm := FALSE;
   XVS_036.CMD.Reset := FALSE;
   XVS_036.CMD.Sim := FALSE;
   XVS_036.CMD.Vector := FALSE;
   XVS_036.CMD.Ready := FALSE;
   XVS_036.CMD.Resourse := FALSE;
   Z_GVM_x.CMD.Hand := FALSE;
   Z_GVM_x.CMD.Start_A := FALSE;
   Z_GVM_x.CMD.Start_M := FALSE;
   Z_GVM_x.CMD.Force := FALSE;
   Z_GVM_x.CMD.Lock := FALSE;
   Z_GVM_x.CMD.Local := FALSE;
   Z_GVM_x.CMD.Service := FALSE;
   Z_GVM_x.CMD.Safety := FALSE;
   Z_GVM_x.CMD.Alarm := FALSE;
   Z_GVM_x.CMD.Reset := FALSE;
   Z_GVM_x.CMD.Sim := FALSE;
   Z_GVM_x.CMD.Vector := FALSE;
   Z_GVM_x.CMD.Ready := FALSE;
   Z_GVM_x.CMD.Resourse := FALSE;
   Z_GVM_x.Status := 0;
   Z_GVM_x.T_ON := 0;
   Z_GVM_x.T_OFF := 0;
   Z_GVM_x.Alarms := 16#0000;
   M_Vent.CMD.Hand := FALSE;
   M_Vent.CMD.Start_A := FALSE;
   M_Vent.CMD.Start_M := FALSE;
   M_Vent.CMD.Force := FALSE;
   M_Vent.CMD.Lock := FALSE;
   M_Vent.CMD.Local := FALSE;
   M_Vent.CMD.Service := FALSE;
   M_Vent.CMD.Safety := FALSE;
   M_Vent.CMD.Alarm := FALSE;
   M_Vent.CMD.Reset := FALSE;
   M_Vent.CMD.Sim := FALSE;
   M_Vent.CMD.Vector := FALSE;
   M_Vent.CMD.Ready := FALSE;
   M_Vent.CMD.Resourse := FALSE;
   M_Vent.Status := 0;
   M_Vent.T_ON := 2;
   M_Vent.T_OFF := 2;
   M_Vent.Alarms := 16#0000;
   M_Vent.Res_h := 9;
   Lines[1..7].Alarms := 16#0000;
END_DATA_BLOCK
